// TwinCAT 3 PLC project Absolute_example
// ProgramVersion: 3.1.4024.0
// libraries:
//   Tc2_MC2, * (Beckhoff Automation GmbH)
//   Tc2_Standard, * (Beckhoff Automation GmbH)
//   Tc2_System, * (Beckhoff Automation GmbH)
//   Tc3_Module, * (Beckhoff Automation GmbH)
// project tree:
//   / PlcTask.TcTTO
//   POUs/ FB_Absolute_Example.TcPOU, MAIN.TcPOU
// real-time tasks:
//   TASK PlcTask: cycle T#10ms, priority 20, ADS port 350
// motion (NC):
//   TASK NC-Task 1 SAF: cycle T#2ms, priority 4, ADS port 501
//   TASK NC-Task 1 SVB: cycle T#10ms, priority 8, ADS port 511
//   AXIS Axis 2 (id 2)
//     Dynamic: Acceleration=7354.05, Deceleration=7354.05, Jerk=22062.1
//     Velo: RefSearch=49.02699, RefSync=49.02699, SlowManual=245.13495, FastManual=1470.8097, Fast=4902.699, Maximum=4902.7
//     OtherSettings: AllowMotionCmdToSlave=true
//     encoder EncType=19
//       EncPara: ScaleFactorNumerator=60, ScaleFactorDenominator=1048576, MaxCount=#xffffffff
//     drive DrvType=16
//       DrvPara: MaxCount=#xffffffff, DriveControlDWord=#x00020100
//         Analog: VeloReferenz=5392.9689, VeloScale=71.5255737304688, TorqueSetpointScale=10, ScaleFactorActTorque=0.1
//         TimeComp: TaskDelayCycles=1
//     controller CtrType=1
//       CtrPara: PriorControlFactor=1
//         Observer: BandWidth=20
//   AXIS Axis 3 (id 3)
//     Dynamic: Acceleration=7354.0485, Deceleration=7354.0485, Jerk=22062.1455
//     Velo: RefSearch=49.02699, RefSync=49.02699, SlowManual=245.13495, FastManual=1470.8097, Fast=4902.699, Maximum=4902.699
//     OtherSettings: AllowMotionCmdToSlave=true
//     encoder EncType=19
//       EncPara: ScaleFactorNumerator=60, ScaleFactorDenominator=1048576, MaxCount=#xffffffff
//     drive DrvType=16
//       DrvPara: MaxCount=#xffffffff, DriveControlDWord=#x00020100
//         Analog: VeloReferenz=5392.9689, VeloScale=71.5255737304688, TorqueSetpointScale=10, ScaleFactorActTorque=0.1
//         TimeComp: TaskDelayCycles=1
//     controller CtrType=1
//       CtrPara: PriorControlFactor=1
//         Observer: BandWidth=20
// I/O:
//   DEVICE Device 1 (EtherCAT), AmsNetId 192.168.98.99.2.1
//     Term 1 (EK1200) [EK1200-5000 EtherCAT Power supply (2A E-Bus)]
//       Term 2 (EL1004) [EL1004 4Ch. Dig. Input 24V, 3ms]
//       Term 3 (EL2004) [EL2004 4Ch. Dig. Output 24V, 0.5A]
//       Term 4 (EL3062) [EL3062 2Ch. Ana. Input 0-10V]
//       Term 5 (EL4002) [EL4002 2Ch. Ana. Output 0-10V, 12bit]
//       Term 6 (EL2008) [EL2008 8Ch. Dig. Output 24V, 0.5A]
//       Term 7 (EK1110) [EK1110 EtherCAT extension]
//     Term 8 (AX8620-0000-0103) [AX8620-0000-0103]
//       Drive 9 (AX8206-0100-0103) [AX8206-0100-0103]
//         modules: Device, Device, Device, Device, Device, Device, Device, Device, Device, Device, Device (Safety), Device, Device, Device, Device, Device, Device, Device, Device, Device, Device, Device, Device, Device, Device, Device, Device, Device, Device, Device, Device, Ch A, Ch A, Ch A, Ch A, Ch A, Ch A, Ch A, Ch A, Ch A, Ch A, Ch A, Ch A, Ch A, Ch A, Ch A, Ch A, Ch A, Ch A, Ch A, Ch A, Ch A, Ch A, Ch A, Ch A, Ch A, Ch A, Ch A, Ch B, Ch B, Ch B, Ch B, Ch B, Ch B, Ch B, Ch B, Ch B, Ch B, Ch B, Ch B, Ch B, Ch B, Ch B, Ch B, Ch B, Ch B, Ch B, Ch B, Ch B, Ch B, Ch B, Ch B, Ch B, Ch B, Ch B
//         startup 12992:1 := 414D383032312D78427830 // Ch A Motor parameters / Configured motor type
//         startup 24768:0 := FEFF // Ch A Interpolation sub mode select
//         startup 13000:5 := 0200 // Ch A Motor thermal model / Reaction
//         startup 13000:6 := 0000C841 // Ch A Motor thermal model / Partial fraction factor
//         startup 12992:12 := 0000FA45 // Ch A Motor parameters / Motor rated speed
//         startup 12992:13 := C9E5FF3E // Ch A Motor parameters / Motor rated torque
//         startup 24694:0 := F4010000 // Ch A Motor standstill torque
//         startup 24800:0 := D007 // Ch A Positive torque/force limit value
//         startup 24801:0 := D007 // Ch A Negative torque/force limit value
//         startup 12288:6 := 4158383230362D303130302D30303030 // Ch A AxisMain parameters / Configured drive type
//         startup 12867:1 := 9A99593F // Ch A TorqueCtrl parameters / Configured channel rated current
//         startup 12867:2 := 33332340 // Ch A TorqueCtrl parameters / Configured channel peak current
//         startup 24672:0 := 08 // Ch A Modes of operation
//         startup 12864:1 := 0D4D7043 // Ch A TorqueCtrl parameters mappable / Torque control proportional gain q
//         startup 12864:2 := 8A0E7C39 // Ch A TorqueCtrl parameters mappable / Torque control integral action time q
//         startup 12608:1 := FBD1CD3B // Ch A VeloCtrl parameters mappable / Velocity control proportional gain
//         startup 12608:2 := 6F12033C // Ch A VeloCtrl parameters mappable / Velocity control integral action time
//         startup 12608:3 := 00980546 // Ch A VeloCtrl parameters mappable / Bipolar velocity limit value
//         startup 12992:15 := 0100 // Ch A Motor parameters / Motor temperature sensor connection
//         startup 12611:4 := 0100 // Ch A VeloCtrl observer / Observer type
//         startup 24672:0 := 08 // Ch A Modes of operation
//         startup 12296:2 := 00 // Ch A AxisMain parameters encoder polarity / Primary encoder actual values
//         startup 14016:1 := 414D383032312D78427830 // Ch B Motor parameters / Configured motor type
//         startup 26816:0 := FEFF // Ch B Interpolation sub mode select
//         startup 14024:5 := 0200 // Ch B Motor thermal model / Reaction
//         startup 14024:6 := 0000C841 // Ch B Motor thermal model / Partial fraction factor
//         startup 14016:12 := 0000FA45 // Ch B Motor parameters / Motor rated speed
//         startup 14016:13 := C9E5FF3E // Ch B Motor parameters / Motor rated torque
//         startup 26742:0 := F4010000 // Ch B Motor standstill torque
//         startup 26848:0 := D007 // Ch B Positive torque/force limit value
//         startup 26849:0 := D007 // Ch B Negative torque/force limit value
//         startup 13312:6 := 4158383230362D303130302D30303030 // Ch B AxisMain parameters / Configured drive type
//         startup 13891:1 := 9A99593F // Ch B TorqueCtrl parameters / Configured channel rated current
//         startup 13891:2 := 33332340 // Ch B TorqueCtrl parameters / Configured channel peak current
//         startup 26720:0 := 08 // Ch B Modes of operation
//         startup 13888:1 := 0D4D7043 // Ch B TorqueCtrl parameters mappable / Torque control proportional gain q
//         startup 13888:2 := 8A0E7C39 // Ch B TorqueCtrl parameters mappable / Torque control integral action time q
//         startup 13632:1 := FBD1CD3B // Ch B VeloCtrl parameters mappable / Velocity control proportional gain
//         startup 13632:2 := 6F12033C // Ch B VeloCtrl parameters mappable / Velocity control integral action time
//         startup 13632:3 := 00980546 // Ch B VeloCtrl parameters mappable / Bipolar velocity limit value
//         startup 14016:15 := 0100 // Ch B Motor parameters / Motor temperature sensor connection
//         startup 13635:4 := 0100 // Ch B VeloCtrl observer / Observer type
//         startup 26720:0 := 08 // Ch B Modes of operation
//         startup 13320:2 := 00 // Ch B AxisMain parameters encoder polarity / Primary encoder actual values
//       Term 10 (EL9011) [EL9011 End Terminal]
// variable links:
//   Device 1 (EtherCAT) <-> Device 1 (EtherCAT)/Term 8 (AX8620-0000-0103)
//     Term 8 (AX8620-0000-0103)/Drive 9 (AX8206-0100-0103)/Device/DeviceMain Outputs/Power supply controlword <-> PSM Controlword for axis/Controlword for axis
//   NC-Task 1 SAF/Axes/Axis 2 <-> Device 1 (EtherCAT)/Term 8 (AX8620-0000-0103)/Drive 9 (AX8206-0100-0103)
//     Drive/Inputs/In/nDataIn1 <-> Ch A/Ch A PositionControl Inputs/Ch A Following error actual value
//     Drive/Inputs/In/nDcOutputTime <-> InfoData/DcOutputShift
//     Drive/Inputs/In/nState1 <-> Ch A/Ch A AxisMain Inputs/Ch A Statusword
//     Drive/Inputs/In/nState2 <-> Ch A/Ch A AxisMain Inputs/Ch A Statusword @bit 8
//     Drive/Outputs/Out/nCtrl1 <-> Ch A/Ch A AxisMain Outputs/Ch A Controlword
//     Drive/Outputs/Out/nCtrl2 <-> Ch A/Ch A AxisMain Outputs/Ch A Controlword @bit 8
//     Drive/Outputs/Out/nDataOut1 <-> Ch A/Ch A Interpolator Outputs/Ch A Target position
//     Drive/Outputs/Out/nDataOut2 <-> Ch A/Ch A Interpolator Outputs/Ch A Target velocity
//     Enc/Inputs/In/nDataIn1 <-> Ch A/Ch A AxisMain Inputs/Ch A Position actual value
//     Enc/Inputs/In/nDcInputTime <-> InfoData/DcInputShift
//     Enc/Inputs/In/nState2 @bit 5 <-> Ch A/Ch A AxisMain Inputs/Position actual value invalid
//   NC-Task 1 SAF/Axes/Axis 3 <-> Device 1 (EtherCAT)/Term 8 (AX8620-0000-0103)/Drive 9 (AX8206-0100-0103)
//     Drive/Inputs/In/nDataIn1 <-> Ch B/Ch B PositionControl Inputs/Ch B Following error actual value
//     Drive/Inputs/In/nDcOutputTime <-> InfoData/DcOutputShift
//     Drive/Inputs/In/nState1 <-> Ch B/Ch B AxisMain Inputs/Ch B Statusword
//     Drive/Inputs/In/nState2 <-> Ch B/Ch B AxisMain Inputs/Ch B Statusword @bit 8
//     Drive/Outputs/Out/nCtrl1 <-> Ch B/Ch B AxisMain Outputs/Ch B Controlword
//     Drive/Outputs/Out/nCtrl2 <-> Ch B/Ch B AxisMain Outputs/Ch B Controlword @bit 8
//     Drive/Outputs/Out/nDataOut1 <-> Ch B/Ch B Interpolator Outputs/Ch B Target position
//     Drive/Outputs/Out/nDataOut2 <-> Ch B/Ch B Interpolator Outputs/Ch B Target velocity
//     Enc/Inputs/In/nDataIn1 <-> Ch B/Ch B AxisMain Inputs/Ch B Position actual value
//     Enc/Inputs/In/nDcInputTime <-> InfoData/DcInputShift
//     Enc/Inputs/In/nState2 @bit 5 <-> Ch B/Ch B AxisMain Inputs/Position actual value invalid
//   Absolute_example/Absolute_example Instance <-> NC-Task 1 SAF/Axes/Axis 2
//     PlcTask Inputs/MAIN.axis_1.NcToPlc <-> Outputs/ToPlc
//     PlcTask Outputs/MAIN.axis_1.PlcToNc <-> Inputs/FromPlc
//   Absolute_example/Absolute_example Instance <-> NC-Task 1 SAF/Axes/Axis 3
//     PlcTask Inputs/MAIN.Axis1.NcToPlc <-> Outputs/ToPlc
//     PlcTask Outputs/MAIN.Axis1.PlcToNc <-> Inputs/FromPlc

CONFIGURATION Absolute_example
    RESOURCE PLC ON TwinCAT3
        TASK PlcTask(INTERVAL := T#10ms, PRIORITY := 20);
        PROGRAM MAIN WITH PlcTask : MAIN;
    END_RESOURCE
END_CONFIGURATION

// ---- POUs/MAIN.TcPOU
PROGRAM MAIN
VAR
	axis_1:		AXIS_REF;
	FBEnable: MC_Power;
	bEnable : BOOL;
	FBAbsolute: MC_MoveAbsolute;
	bAbsolute : BOOL;
	
	fb_absolute_Example    : FB_Absolute_Example;
	Axis1: AXIS_REF;
	fPosition1:		 LREAL;
	fPosition2:		 LREAL;
	fPosition3		:LREAL;
	tDelay: 		 TIME;
	fVelocity:		 LREAL;
	bError:			 BOOL;
	sStatus:		 STRING;
	
	bBool			:BOOL;
	bBool1: INT;
	fb_Reset: MC_Reset;
	
	
   
    bBoool	:		BOOL;
	position	:	LREAL;
	mode		:	BOOL;
	options		:ST_SetPositionOptions;
	fb_SetPosition: MC_SetPosition;
END_VAR



fb_absolute_Example(
	bEnable:=bEnable , 
	fPosition1:= fPosition1, 
	fPosition2:=fPosition2 , 
	fPosition3:= fPosition3, 
	tDelay:= tDelay, 
	fVelocity:= fVelocity, 
	bError=>bError , 
	sStatus=>sStatus , 
	Axis:=axis_1 );

END_PROGRAM

// ---- POUs/FB_Absolute_Example.TcPOU
FUNCTION_BLOCK FB_Absolute_Example
VAR_INPUT
	bEnable		:BOOL;
	fPosition1	:LREAL;
	fPosition2	:LREAL;
	fPosition3	:LREAL;
	tDelay		:TIME;	
	fVelocity	:LREAL;
	
END_VAR
VAR_OUTPUT
	bError		:BOOL;
	sStatus		:STRING;
END_VAR

VAR
	fb_Power		: MC_Power;
	stateDataFlow	: (RESET_STATE, FIRST_MOVE_STATE, FIRST_MOTION_CONTROL_STATE, FIRST_WAIT_STATE, 
SECOND_MOVE_STATE, SECOND_MOTION_CONTROL_STATE, SECOND_WAIT_STATE, THIRD_MOVE_STATE,THIRD_MOTION_CONTROL_STATE,THIRD_WAIT_STATE, ERROR_STATE):=RESET_STATE;
	fbTimer			:TON;	
	fb_MoveAbsolute: MC_MoveAbsolute;
END_VAR
VAR_IN_OUT
	Axis :		AXIS_REF;
END_VAR


fbTimer(PT:=tDelay);

CASE stateDataFlow OF
	
RESET_STATE:
		bError			:=FALSE;
		sStatus			:='Beklemede';
		
		IF bEnable THEN
			stateDataFlow:=FIRST_MOVE_STATE;
			ELSIF NOT Axis.Status.Operational THEN
				stateDataFlow:=ERROR_STATE;
				sStatus:='Enable değil';
		END_IF
	fb_Power(
	Axis:= Axis, 
	Enable:=bEnable , 
	Enable_Positive:= bEnable, 
	Enable_Negative:=bEnable , 
	Override:=100 ,);
	

FIRST_MOVE_STATE:
	
	fb_MoveAbsolute.Position:=fPosition1;
	fb_MoveAbsolute.Execute 	:= TRUE;
	IF Axis.Status.Moving THEN 
		stateDataFlow:=FIRST_MOTION_CONTROL_STATE;
		sStatus:= '1. Noktaya gidiyor';
		ELSIF Axis.Status.Error OR fb_MoveAbsolute.Error THEN
		
		sStatus		:='1. noktaya giderken hataya geçti'	;
		stateDataFlow:=ERROR_STATE;
		
	END_IF 
	
FIRST_MOTION_CONTROL_STATE:
	IF fb_MoveAbsolute.Done THEN 
			stateDataFlow:=FIRST_WAIT_STATE;
			fb_MoveAbsolute.Execute:=FALSE;
		END_IF
	
FIRST_WAIT_STATE:

		fbTimer.IN:=TRUE;
		sStatus		:='1. noktada bekliyor ';
		
		IF fbTimer.Q THEN 
			fbTimer.IN:=FALSE;
			stateDataFlow:=SECOND_MOVE_STATE;
		END_IF	
		
SECOND_MOVE_STATE	:

	fb_MoveAbsolute.Position:=fPosition2;
	fVelocity:=fVelocity/2;
			fb_MoveAbsolute.Execute 	:= TRUE;
			IF Axis.Status.Moving THEN 
				
				stateDataFlow:=SECOND_MOTION_CONTROL_STATE;
				sStatus:= '2. Noktaya gidiyor';
				ELSIF Axis.Status.Error OR fb_MoveAbsolute.Error THEN
				
				sStatus		:='2. noktaya giderken hataya geçti';
				stateDataFlow:=ERROR_STATE;
			END_IF

SECOND_MOTION_CONTROL_STATE:
			
		IF fb_MoveAbsolute.Done THEN
			stateDataFlow := SECOND_WAIT_STATE;
			fb_MoveAbsolute.Execute:=FALSE;
			 
		END_IF
		
SECOND_WAIT_STATE:
	fbTimer.IN:=TRUE;
		
		sStatus		:='2. noktada bekliyor ';
		
		IF fbTimer.Q THEN 
			fbTimer.IN:=FALSE;
			stateDataFlow:=THIRD_MOVE_STATE;
		END_IF

		
		
		
THIRD_MOVE_STATE	:	

	fb_MoveAbsolute.Position:=fposition3;
	
			fb_MoveAbsolute.Execute 	:= TRUE;
			IF Axis.Status.Moving THEN 
				
				stateDataFlow:=THIRD_MOTION_CONTROL_STATE;
				sStatus:= '3. Noktaya gidiyor';
				ELSIF Axis.Status.Error OR fb_MoveAbsolute.Error THEN
				
				sStatus		:='3. noktaya giderken hataya geçti';
				stateDataFlow:=ERROR_STATE;
			END_IF

			
THIRD_MOTION_CONTROL_STATE:
	
	IF fb_MoveAbsolute.Done THEN
			stateDataFlow := THIRD_WAIT_STATE;
			fb_MoveAbsolute.Execute:=FALSE;
			 
		END_IF

				
THIRD_WAIT_STATE:
	fbTimer.IN:=TRUE;
		sStatus		:='3. noktada bekliyor ';
		
		IF fbTimer.Q THEN 
			fbTimer.IN:=FALSE;
			stateDataFlow:=RESET_STATE;
		END_IF

		
ERROR_STATE:
	bError :=FALSE;
		
		IF NOT bEnable THEN
			fbTimer(IN:= FALSE);
			stateDataFlow:=RESET_STATE;
		END_IF

	END_CASE

fb_MoveAbsolute(
	Axis:= Axis, 
	Velocity:=fVelocity ,);
	Axis.ReadStatus();

END_FUNCTION_BLOCK
